(* CODESYS project Machine.xml

Project tree, tasks and I/O mapping:
  program Machine [CFC]
*)

// Machine
PROGRAM Machine
VAR
	Sequence: 			BagFeedSequence;	//
END_VAR
VAR // added by the converter: edge detectors and wires of the graphical bodies
    _w1 : ANY;
END_VAR

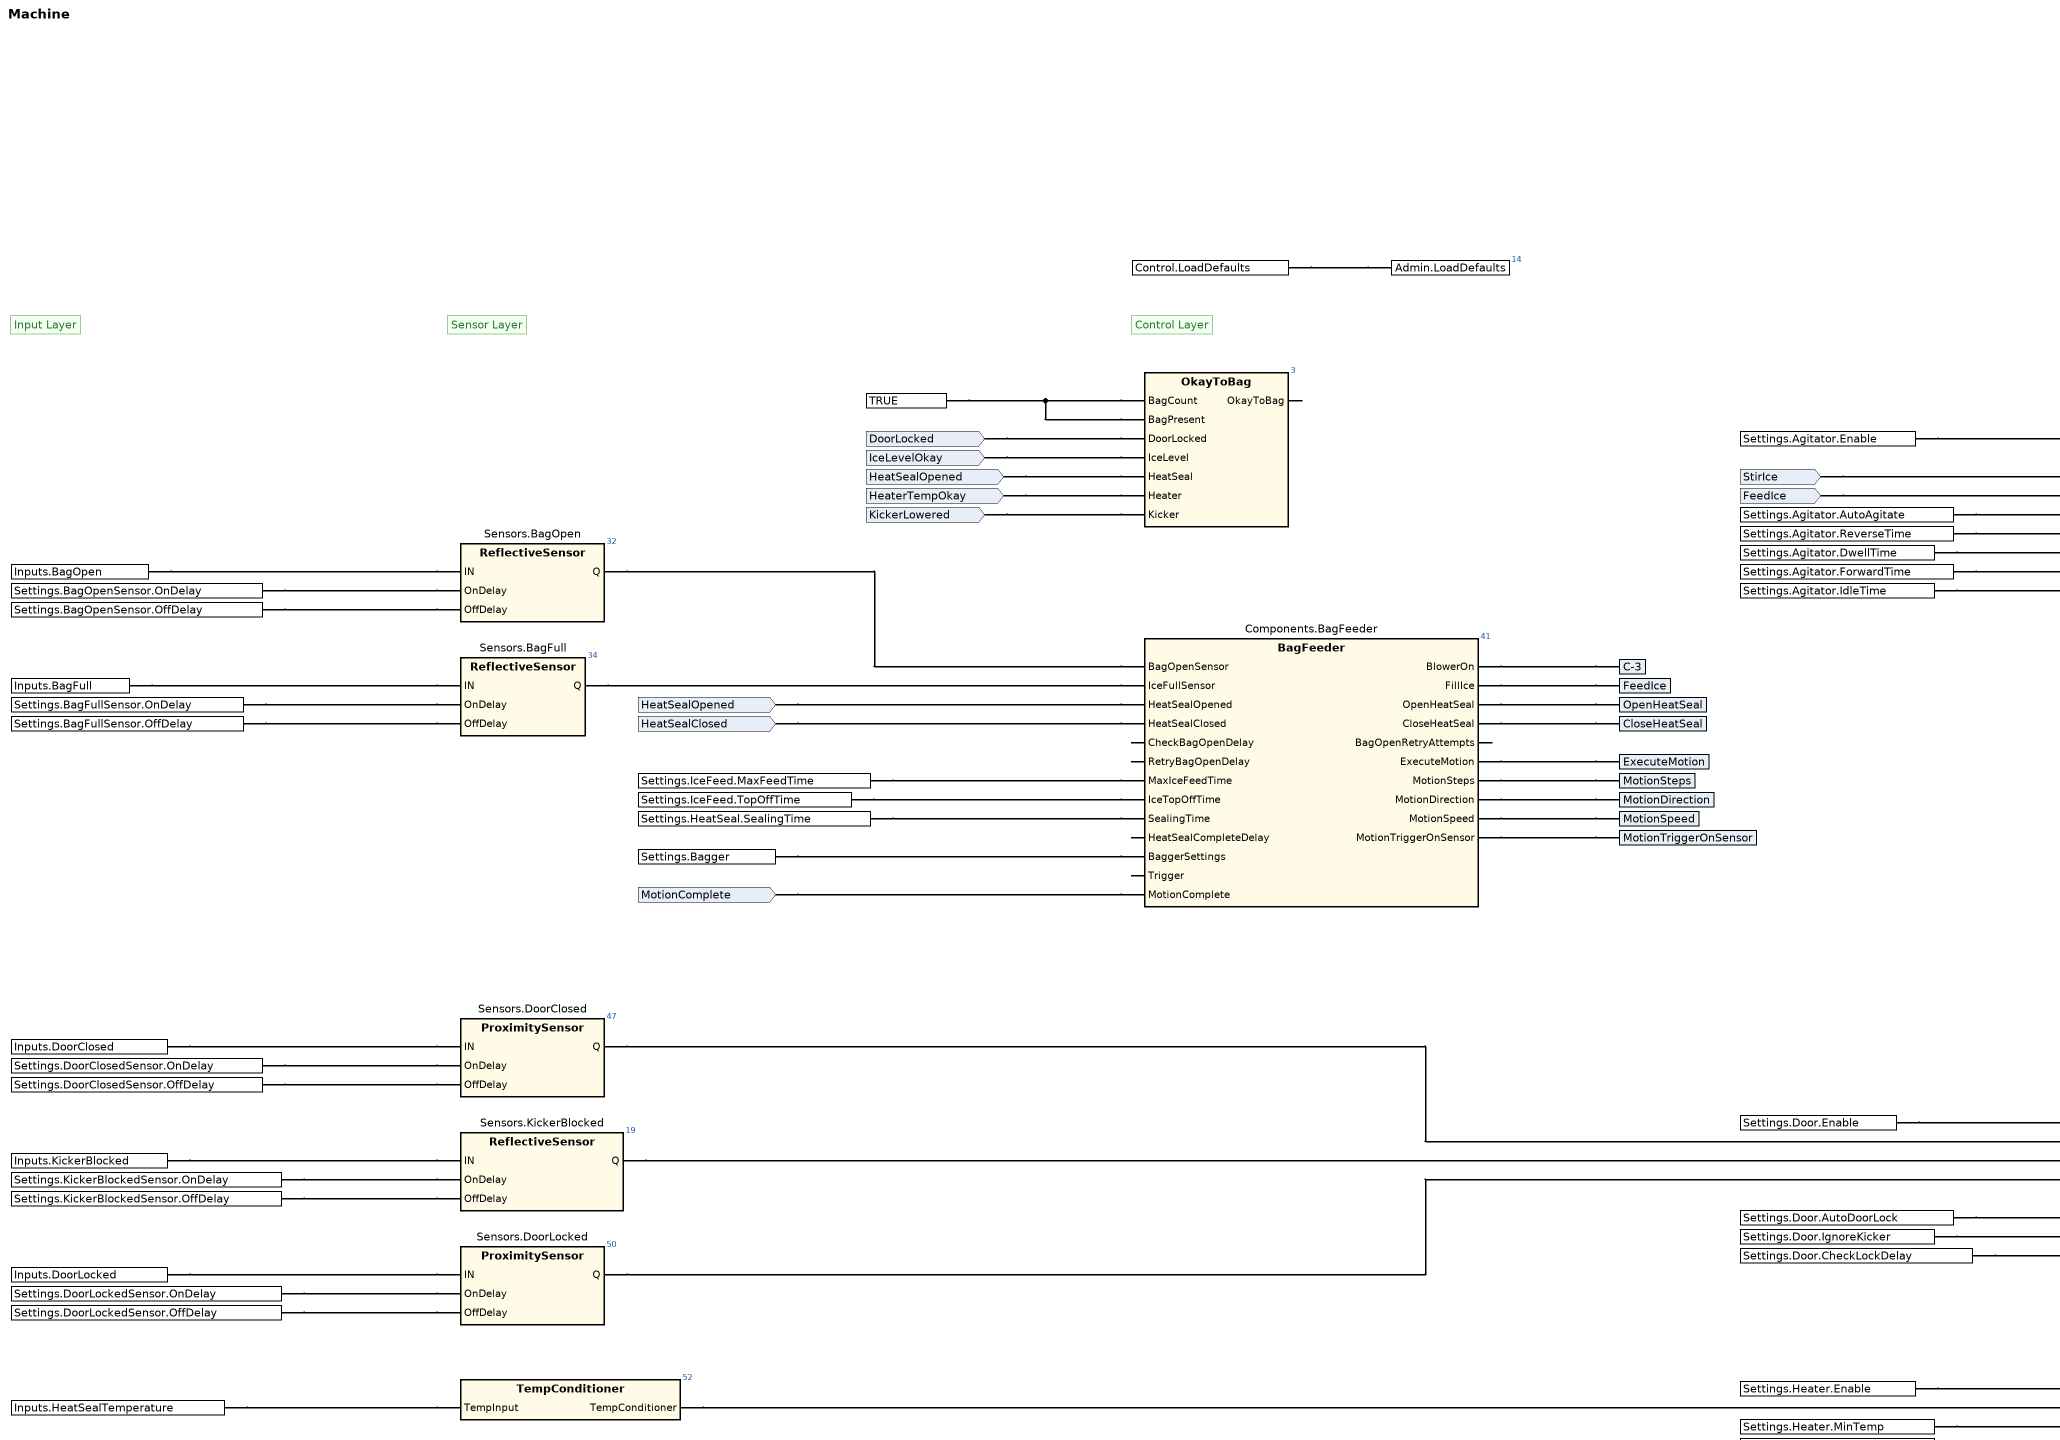
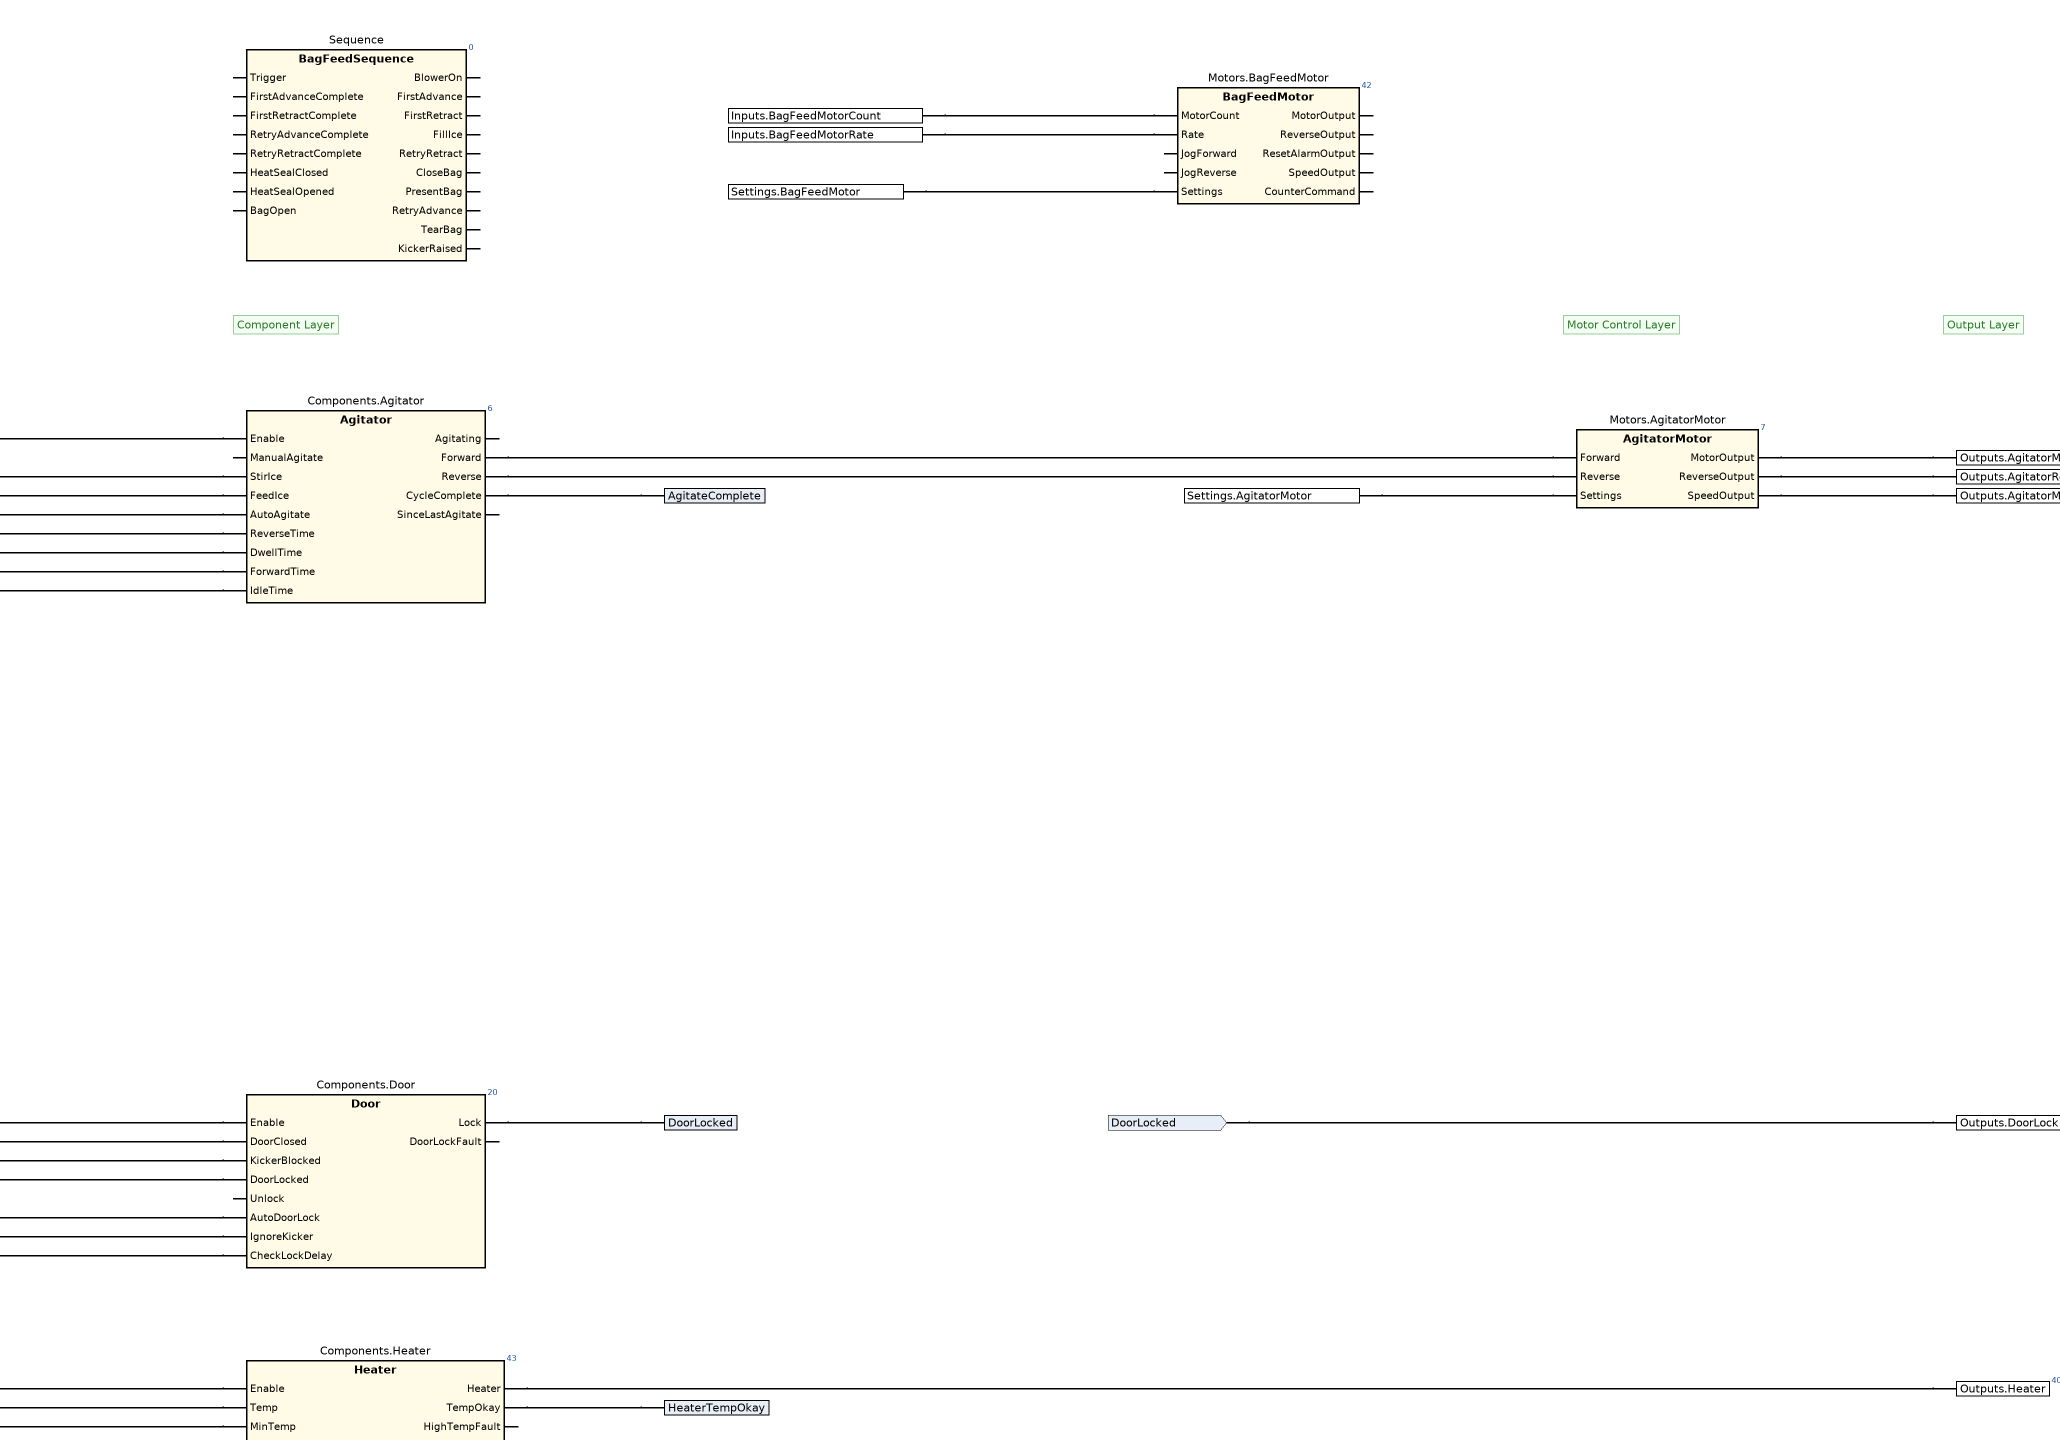
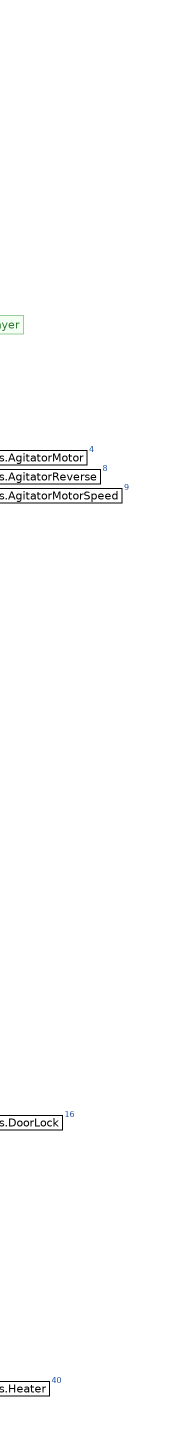
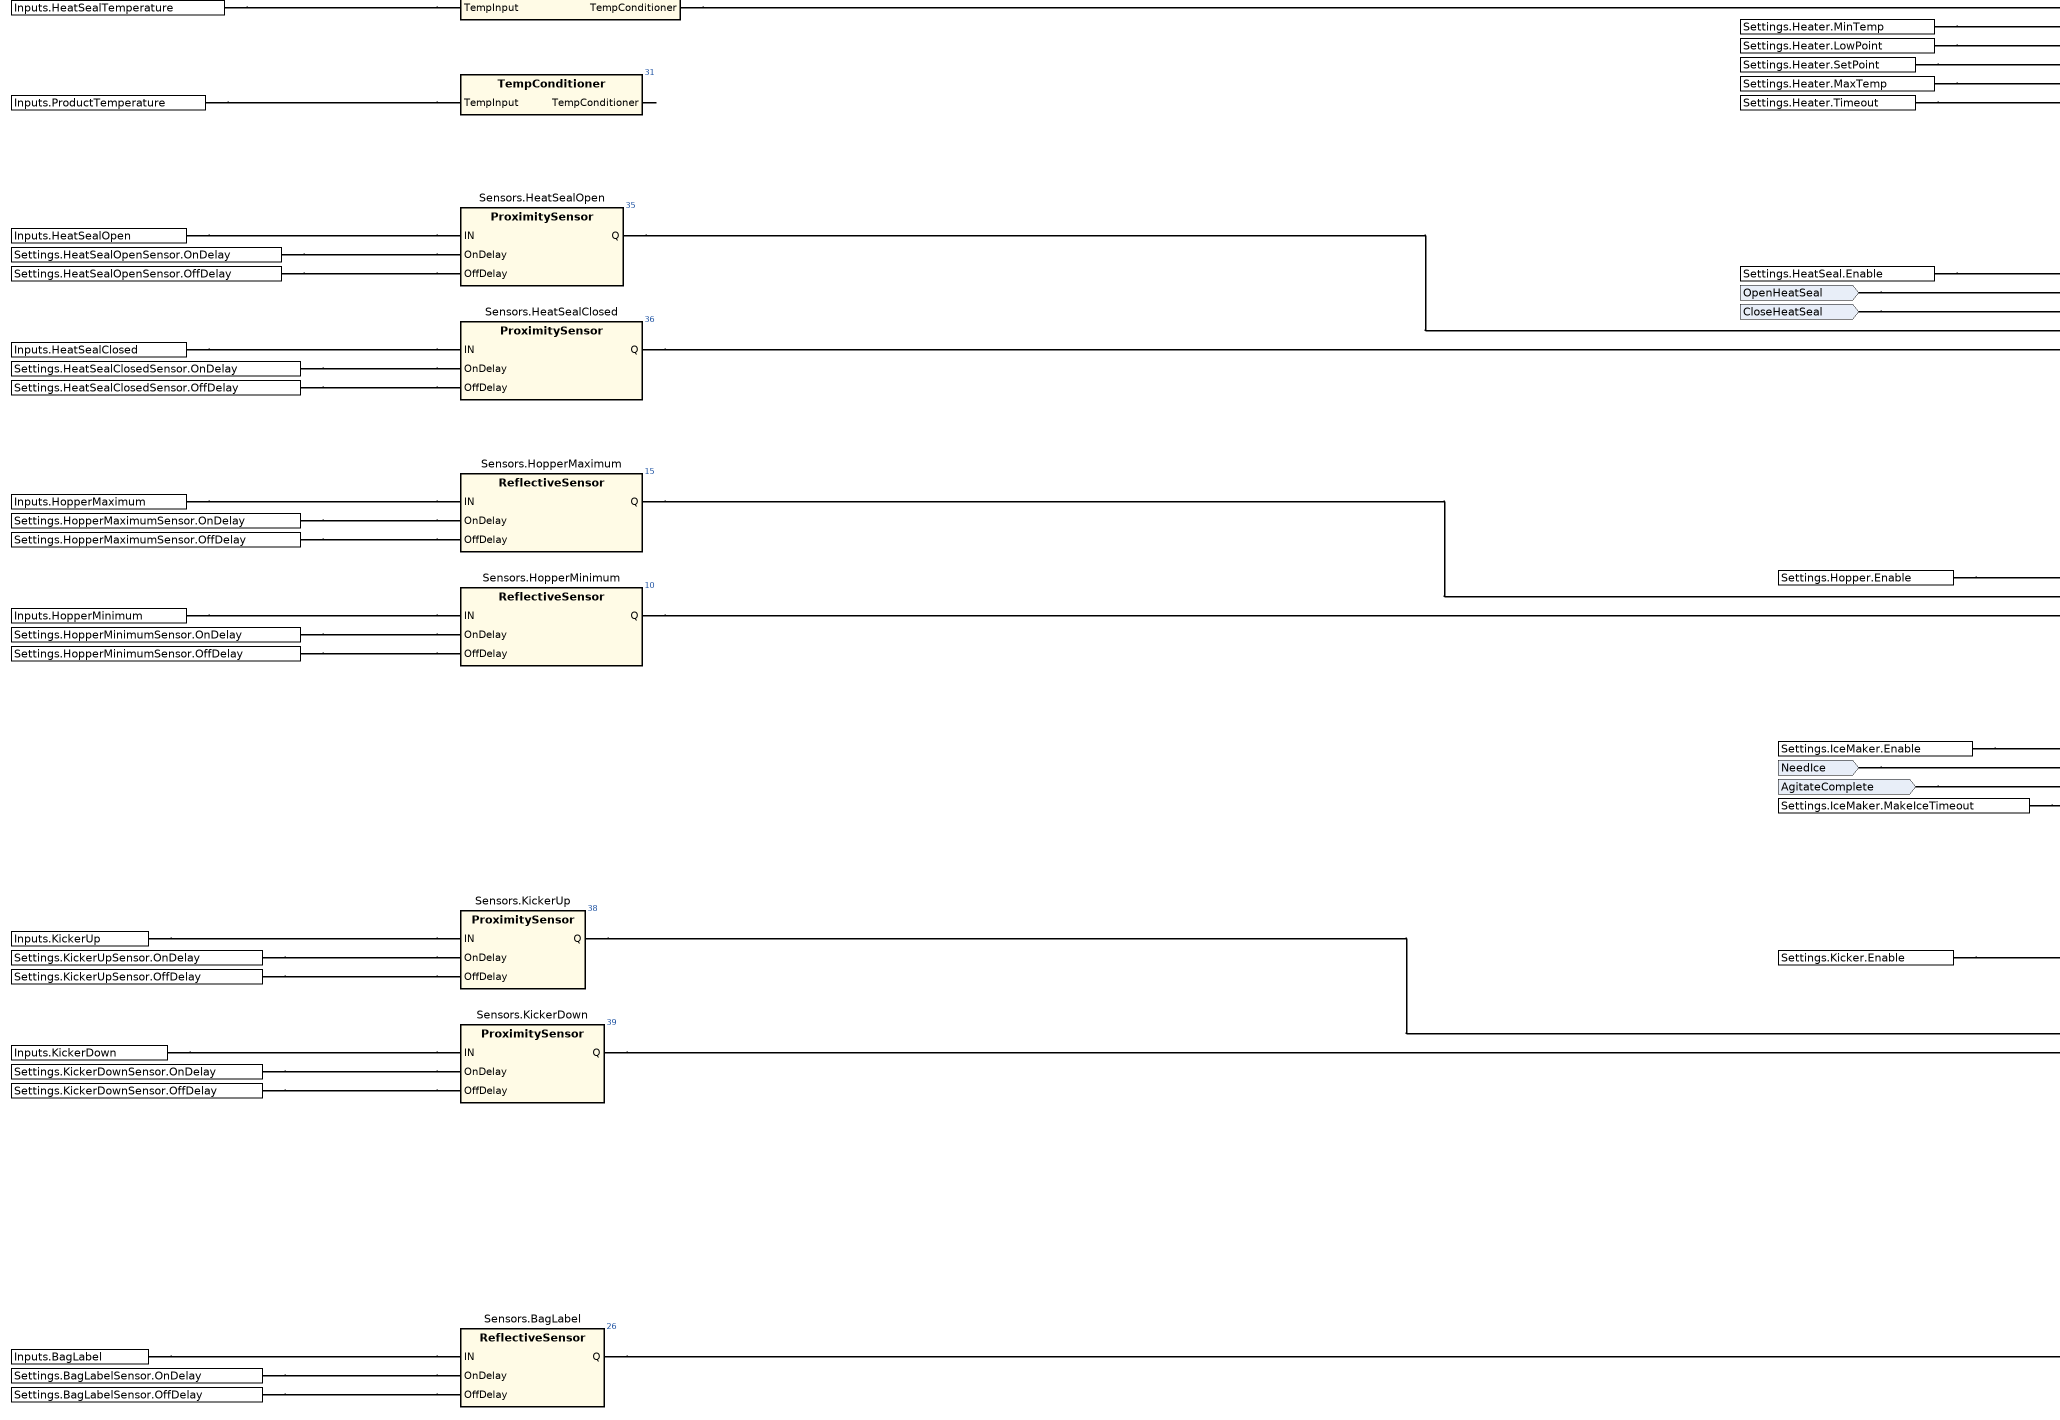
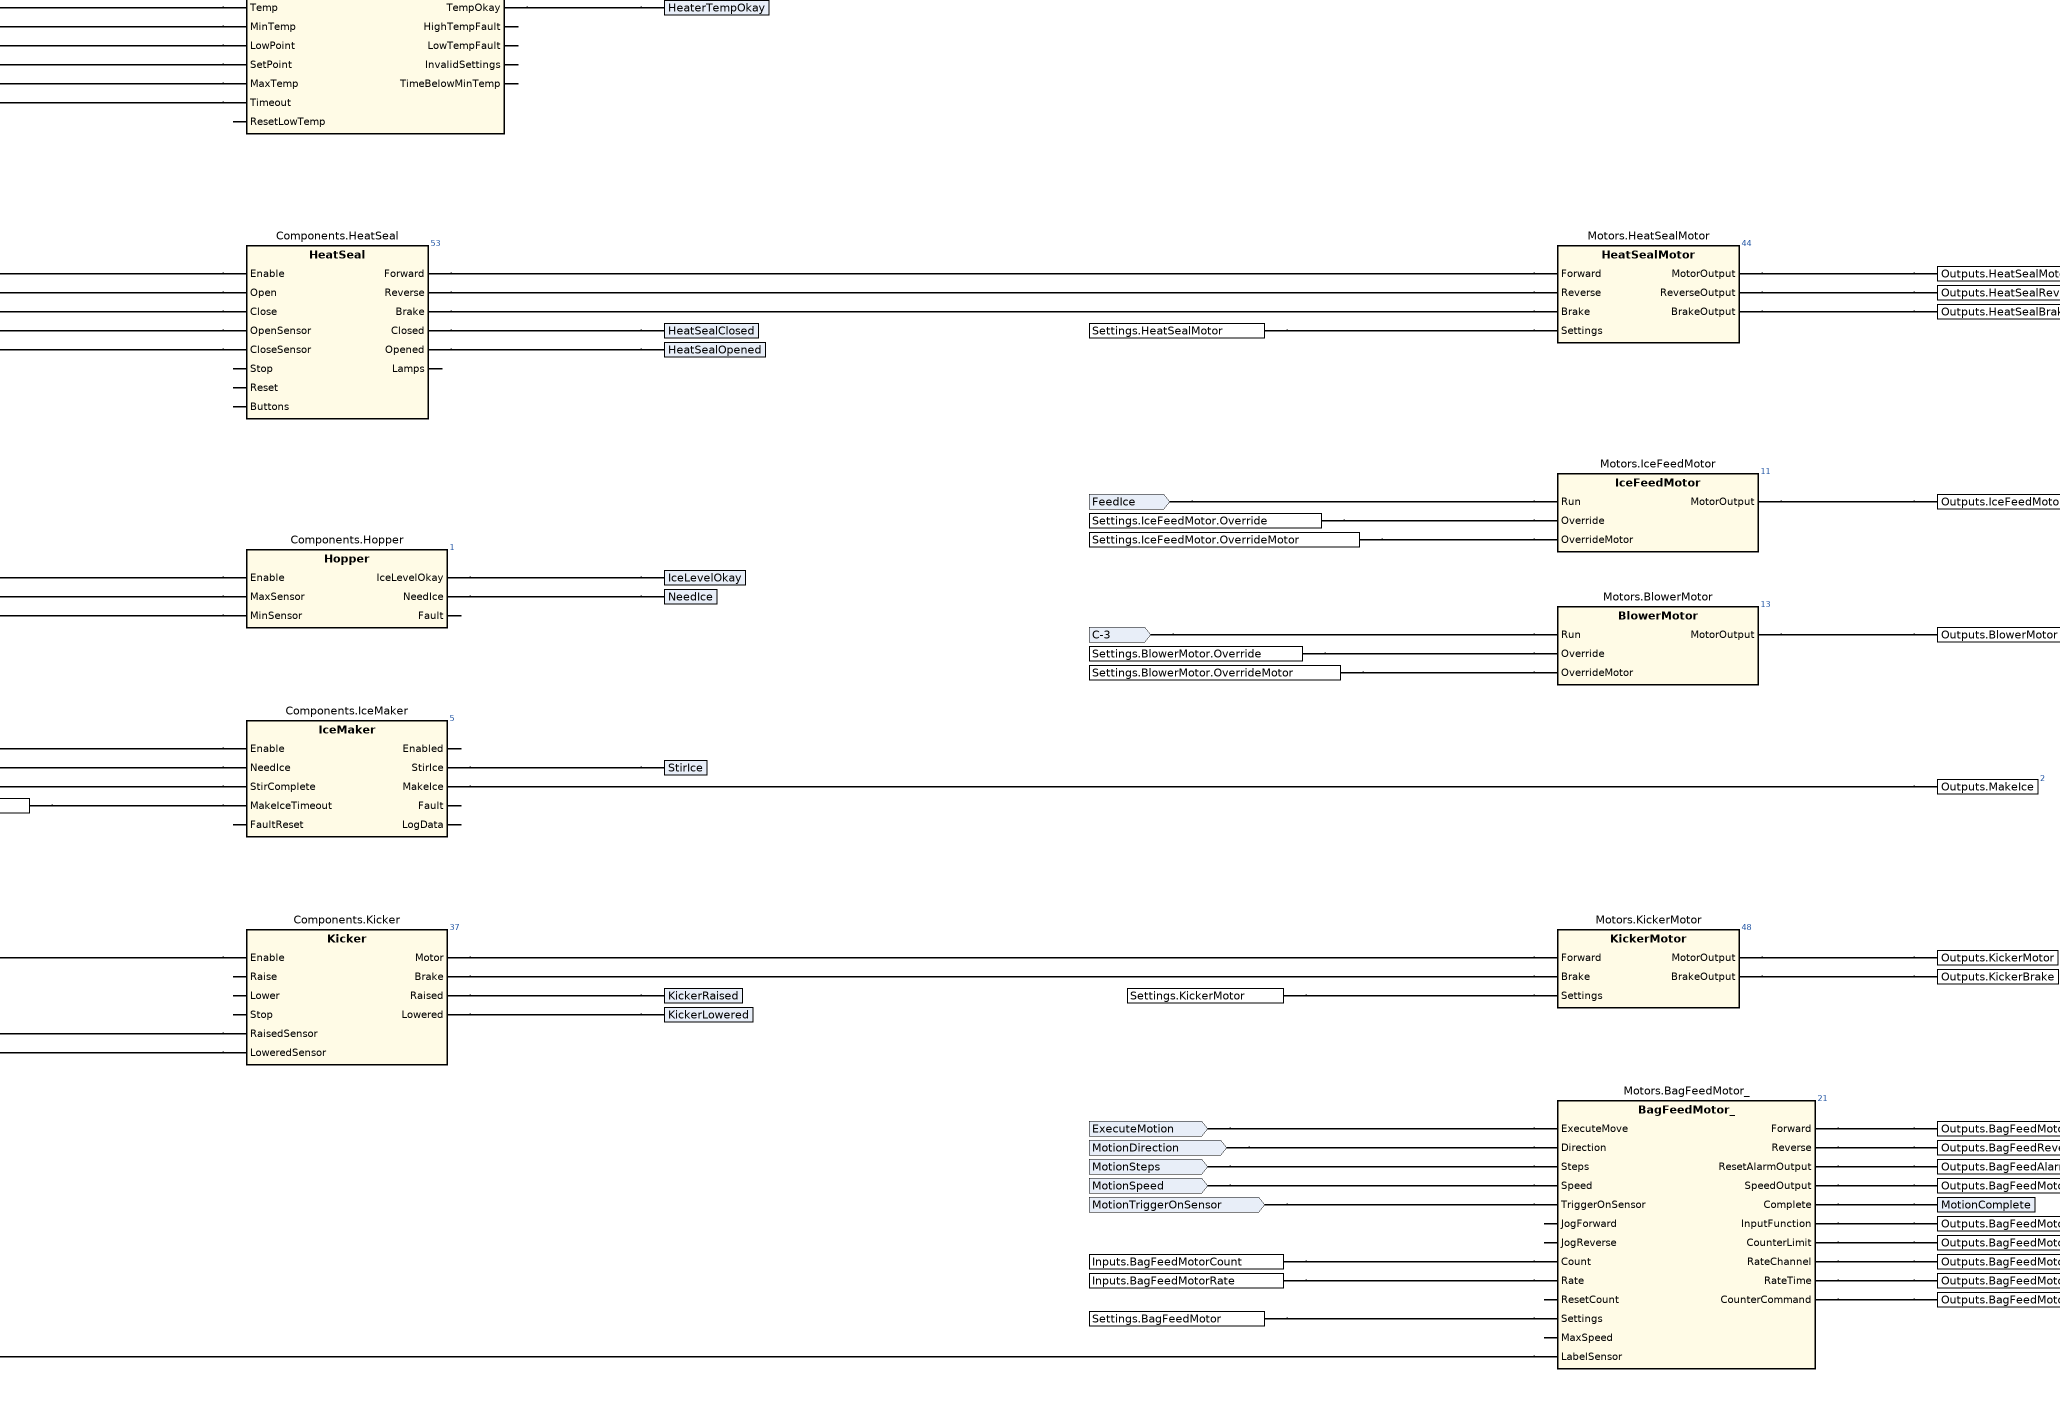
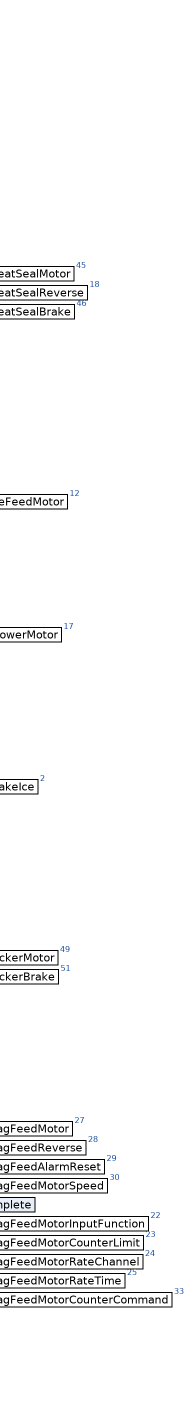
// note: 5 stored wires end on pins the file does not list and are not shown
Sequence(); // BagFeedSequence
Components.Hopper(
    Enable := Settings.Hopper.Enable,
    MaxSensor := Sensors.HopperMaximum.Q,
    MinSensor := Sensors.HopperMinimum.Q); // Hopper
Outputs.MakeIce := Components.IceMaker.MakeIce;
// Control Layer
OkayToBag(BagCount := TRUE, BagPresent := TRUE, DoorLocked := Components.Door.Lock, IceLevel := Components.Hopper.IceLevelOkay, HeatSeal := Components.HeatSeal.Opened, Heater := Components.Heater.TempOkay, Kicker := Components.Kicker.Lowered);
// Output Layer
Outputs.AgitatorMotor := Motors.AgitatorMotor.MotorOutput;
Components.IceMaker(
    Enable := Settings.IceMaker.Enable,
    NeedIce := Components.Hopper.NeedIce,
    StirComplete := Components.Agitator.CycleComplete,
    MakeIceTimeout := Settings.IceMaker.MakeIceTimeout); // IceMaker
// Component Layer
Components.Agitator(
    Enable := Settings.Agitator.Enable,
    StirIce := Components.IceMaker.StirIce,
    FeedIce := Components.BagFeeder.FillIce,
    AutoAgitate := Settings.Agitator.AutoAgitate,
    ReverseTime := Settings.Agitator.ReverseTime,
    DwellTime := Settings.Agitator.DwellTime,
    ForwardTime := Settings.Agitator.ForwardTime,
    IdleTime := Settings.Agitator.IdleTime); // Agitator
// Motor Control Layer
Motors.AgitatorMotor(
    Forward := Components.Agitator.Forward,
    Reverse := Components.Agitator.Reverse,
    Settings := Settings.AgitatorMotor); // AgitatorMotor
Outputs.AgitatorReverse := Motors.AgitatorMotor.ReverseOutput;
Outputs.AgitatorMotorSpeed := Motors.AgitatorMotor.SpeedOutput;
Sensors.HopperMinimum(
    IN := Inputs.HopperMinimum,
    OnDelay := Settings.HopperMinimumSensor.OnDelay,
    OffDelay := Settings.HopperMinimumSensor.OffDelay); // ReflectiveSensor
Motors.IceFeedMotor(
    Run := Components.BagFeeder.FillIce,
    Override := Settings.IceFeedMotor.Override,
    OverrideMotor := Settings.IceFeedMotor.OverrideMotor); // IceFeedMotor
Outputs.IceFeedMotor := Motors.IceFeedMotor.MotorOutput;
Motors.BlowerMotor(
    Run := Components.BagFeeder.BlowerOn,
    Override := Settings.BlowerMotor.Override,
    OverrideMotor := Settings.BlowerMotor.OverrideMotor); // BlowerMotor
Admin.LoadDefaults := Control.LoadDefaults;
Sensors.HopperMaximum(
    IN := Inputs.HopperMaximum,
    OnDelay := Settings.HopperMaximumSensor.OnDelay,
    OffDelay := Settings.HopperMaximumSensor.OffDelay); // ReflectiveSensor
Outputs.DoorLock := Components.Door.Lock;
Outputs.BlowerMotor := Motors.BlowerMotor.MotorOutput;
Outputs.HeatSealReverse := Motors.HeatSealMotor.ReverseOutput;
Sensors.KickerBlocked(
    IN := Inputs.KickerBlocked,
    OnDelay := Settings.KickerBlockedSensor.OnDelay,
    OffDelay := Settings.KickerBlockedSensor.OffDelay); // ReflectiveSensor
Components.Door(
    Enable := Settings.Door.Enable,
    DoorClosed := Sensors.DoorClosed.Q,
    KickerBlocked := Sensors.KickerBlocked.Q,
    DoorLocked := Sensors.DoorLocked.Q,
    AutoDoorLock := Settings.Door.AutoDoorLock,
    IgnoreKicker := Settings.Door.IgnoreKicker,
    CheckLockDelay := Settings.Door.CheckLockDelay); // Door
Motors.BagFeedMotor_(
    ExecuteMove := Components.BagFeeder.ExecuteMotion,
    Direction := Components.BagFeeder.MotionDirection,
    Steps := Components.BagFeeder.MotionSteps,
    Speed := Components.BagFeeder.MotionSpeed,
    TriggerOnSensor := Components.BagFeeder.MotionTriggerOnSensor,
    Count := Inputs.BagFeedMotorCount,
    Rate := Inputs.BagFeedMotorRate,
    Settings := Settings.BagFeedMotor,
    LabelSensor := Sensors.BagLabel.Q); // BagFeedMotor_
Outputs.BagFeedMotorInputFunction := Motors.BagFeedMotor_.InputFunction;
Outputs.BagFeedMotorCounterLimit := Motors.BagFeedMotor_.CounterLimit;
Outputs.BagFeedMotorRateChannel := Motors.BagFeedMotor_.RateChannel;
Outputs.BagFeedMotorRateTime := Motors.BagFeedMotor_.RateTime;
Sensors.BagLabel(
    IN := Inputs.BagLabel,
    OnDelay := Settings.BagLabelSensor.OnDelay,
    OffDelay := Settings.BagLabelSensor.OffDelay); // ReflectiveSensor
Outputs.BagFeedMotor := Motors.BagFeedMotor_.Forward;
Outputs.BagFeedReverse := Motors.BagFeedMotor_.Reverse;
Outputs.BagFeedAlarmReset := Motors.BagFeedMotor_.ResetAlarmOutput;
Outputs.BagFeedMotorSpeed := Motors.BagFeedMotor_.SpeedOutput;
TempConditioner(TempInput := Inputs.ProductTemperature);
// Input Layer
// Sensor Layer
Sensors.BagOpen(
    IN := Inputs.BagOpen,
    OnDelay := Settings.BagOpenSensor.OnDelay,
    OffDelay := Settings.BagOpenSensor.OffDelay); // ReflectiveSensor
Outputs.BagFeedMotorCounterCommand := Motors.BagFeedMotor_.CounterCommand;
Sensors.BagFull(
    IN := Inputs.BagFull,
    OnDelay := Settings.BagFullSensor.OnDelay,
    OffDelay := Settings.BagFullSensor.OffDelay); // ReflectiveSensor
Sensors.HeatSealOpen(
    IN := Inputs.HeatSealOpen,
    OnDelay := Settings.HeatSealOpenSensor.OnDelay,
    OffDelay := Settings.HeatSealOpenSensor.OffDelay); // ProximitySensor
Sensors.HeatSealClosed(
    IN := Inputs.HeatSealClosed,
    OnDelay := Settings.HeatSealClosedSensor.OnDelay,
    OffDelay := Settings.HeatSealClosedSensor.OffDelay); // ProximitySensor
Components.Kicker(
    Enable := Settings.Kicker.Enable,
    RaisedSensor := Sensors.KickerUp.Q,
    LoweredSensor := Sensors.KickerDown.Q); // Kicker
Sensors.KickerUp(
    IN := Inputs.KickerUp,
    OnDelay := Settings.KickerUpSensor.OnDelay,
    OffDelay := Settings.KickerUpSensor.OffDelay); // ProximitySensor
Sensors.KickerDown(
    IN := Inputs.KickerDown,
    OnDelay := Settings.KickerDownSensor.OnDelay,
    OffDelay := Settings.KickerDownSensor.OffDelay); // ProximitySensor
Outputs.Heater := Components.Heater.Heater;
Components.BagFeeder(
    BagOpenSensor := Sensors.BagOpen.Q,
    IceFullSensor := Sensors.BagFull.Q,
    HeatSealOpened := Components.HeatSeal.Opened,
    HeatSealClosed := Components.HeatSeal.Closed,
    MaxIceFeedTime := Settings.IceFeed.MaxFeedTime,
    IceTopOffTime := Settings.IceFeed.TopOffTime,
    SealingTime := Settings.HeatSeal.SealingTime,
    BaggerSettings := Settings.Bagger,
    MotionComplete := Motors.BagFeedMotor_.Complete); // BagFeeder
Motors.BagFeedMotor(
    MotorCount := Inputs.BagFeedMotorCount,
    Rate := Inputs.BagFeedMotorRate,
    Settings := Settings.BagFeedMotor); // BagFeedMotor
Components.Heater(
    Enable := Settings.Heater.Enable,
    Temp := _w1,
    MinTemp := Settings.Heater.MinTemp,
    LowPoint := Settings.Heater.LowPoint,
    SetPoint := Settings.Heater.SetPoint,
    MaxTemp := Settings.Heater.MaxTemp,
    Timeout := Settings.Heater.Timeout); // Heater
Motors.HeatSealMotor(
    Forward := Components.HeatSeal.Forward,
    Reverse := Components.HeatSeal.Reverse,
    Brake := Components.HeatSeal.Brake,
    Settings := Settings.HeatSealMotor); // HeatSealMotor
Outputs.HeatSealMotor := Motors.HeatSealMotor.MotorOutput;
Outputs.HeatSealBrake := Motors.HeatSealMotor.BrakeOutput;
Sensors.DoorClosed(
    IN := Inputs.DoorClosed,
    OnDelay := Settings.DoorClosedSensor.OnDelay,
    OffDelay := Settings.DoorClosedSensor.OffDelay); // ProximitySensor
Motors.KickerMotor(
    Forward := Components.Kicker.Motor,
    Brake := Components.Kicker.Brake,
    Settings := Settings.KickerMotor); // KickerMotor
Outputs.KickerMotor := Motors.KickerMotor.MotorOutput;
Sensors.DoorLocked(
    IN := Inputs.DoorLocked,
    OnDelay := Settings.DoorLockedSensor.OnDelay,
    OffDelay := Settings.DoorLockedSensor.OffDelay); // ProximitySensor
Outputs.KickerBrake := Motors.KickerMotor.BrakeOutput;
_w1 := TempConditioner(TempInput := Inputs.HeatSealTemperature);
Components.HeatSeal(
    Enable := Settings.HeatSeal.Enable,
    Open := Components.BagFeeder.OpenHeatSeal,
    Close := Components.BagFeeder.CloseHeatSeal,
    OpenSensor := Sensors.HeatSealOpen.Q,
    CloseSensor := Sensors.HeatSealClosed.Q); // HeatSeal

END_PROGRAM
